# EPICS substitutions: iocBoot/iocZed/fb_epid.substitutions
# $Id: fb_epid.substitutions 14505 2012-02-29 21:25:07Z jemian $

file "$(OPTICS)/opticsApp/Db/fb_epid.db"
  {
    {
        P=zzz:epid1,
	IN=zzz:epid1:sim.VAL,
	OUT=zzz:epid1:sim.D,
	MODE=PID,
	CALC=A,
	PERMIT1="zzz:epid1:on.VAL",
	PERMIT2="",
	PERMIT3="",
	PERMIT4=""
    }
  }
